(* IEC 61131-3 sources: com.logicals.lc3.webinar/usRTS_RPMControl_iSOC/src_FB_LIB_SAFE/Convert/LWORD, 4 files *)

(* ---- wLWORD_TO_ULINT.iecst ---- *)
NAMESPACE logicals.web.standard
NAMESPACE convert

/*
 * Function block wrapper for IEC 61131-3 TO_ULINT<br>
 * IN =  input value (LWORD)<br>
 * OUT = IN (ULINT)<br>
 */
FUNCTION_BLOCK wLWORD_TO_ULINT
	{ vNameAlignment:="center"; altName:="LWORD_TO_ULINT"; bgColor:="Plum"; width:=140; hideIONames; }
	VAR_INPUT
		IN : LWORD;
	END_VAR
	VAR_OUTPUT
		OUT: ULINT;
	END_VAR

	OUT := TO_ULINT(IN:=IN, ENO=>ENO);
END_FUNCTION_BLOCK

END_NAMESPACE
END_NAMESPACE

(* ---- wTRUNC_LWORD_TO_BYTE.iecst ---- *)
NAMESPACE logicals.web.standard
NAMESPACE convert

/*
 * Function block wrapper for IEC 61131-3 TO_BYTE<br>
 * IN =  input value (LWORD)<br>
 * OUT = IN (BYTE)<br>
 */
FUNCTION_BLOCK wTRUNC_LWORD_TO_BYTE
	{ vNameAlignment:="center"; altName:="TRUNC_LWORD_TO_BYTE"; bgColor:="DodgerBlue"; width:=200; hideIONames; }
	VAR_INPUT
		IN : LWORD;
	END_VAR
	VAR_OUTPUT
		OUT: BYTE;
	END_VAR

	OUT := TO_BYTE(IN:=IN, ENO=>ENO);
END_FUNCTION_BLOCK

END_NAMESPACE
END_NAMESPACE

(* ---- wTRUNC_LWORD_TO_DWORD.iecst ---- *)
NAMESPACE logicals.web.standard
NAMESPACE convert

/*
 * Function block wrapper for IEC 61131-3 TO_DWORD<br>
 * IN =  input value (LWORD)<br>
 * OUT = IN (DWORD)<br>
 */
FUNCTION_BLOCK wTRUNC_LWORD_TO_DWORD
	{ vNameAlignment:="center"; altName:="TRUNC_LWORD_TO_DWORD"; bgColor:="DodgerBlue"; width:=200; hideIONames; }
	VAR_INPUT
		IN : LWORD;
	END_VAR
	VAR_OUTPUT
		OUT: DWORD;
	END_VAR

	OUT := TO_DWORD(IN:=IN, ENO=>ENO);
END_FUNCTION_BLOCK

END_NAMESPACE
END_NAMESPACE

(* ---- wTRUNC_LWORD_TO_WORD.iecst ---- *)
NAMESPACE logicals.web.standard
NAMESPACE convert

/*
 * Function block wrapper for IEC 61131-3 TO_WORD<br>
 * IN =  input value (LWORD)<br>
 * OUT = IN (WORD)<br>
 */
FUNCTION_BLOCK wTRUNC_LWORD_TO_WORD
	{ vNameAlignment:="center"; altName:="TRUNC_LWORD_TO_WORD"; bgColor:="DodgerBlue"; width:=200; hideIONames; }
	VAR_INPUT
		IN : LWORD;
	END_VAR
	VAR_OUTPUT
		OUT: WORD;
	END_VAR

	OUT := TO_WORD(IN:=IN, ENO=>ENO);
END_FUNCTION_BLOCK

END_NAMESPACE
END_NAMESPACE
